RoboDK station: Dexter_ER2.rdk

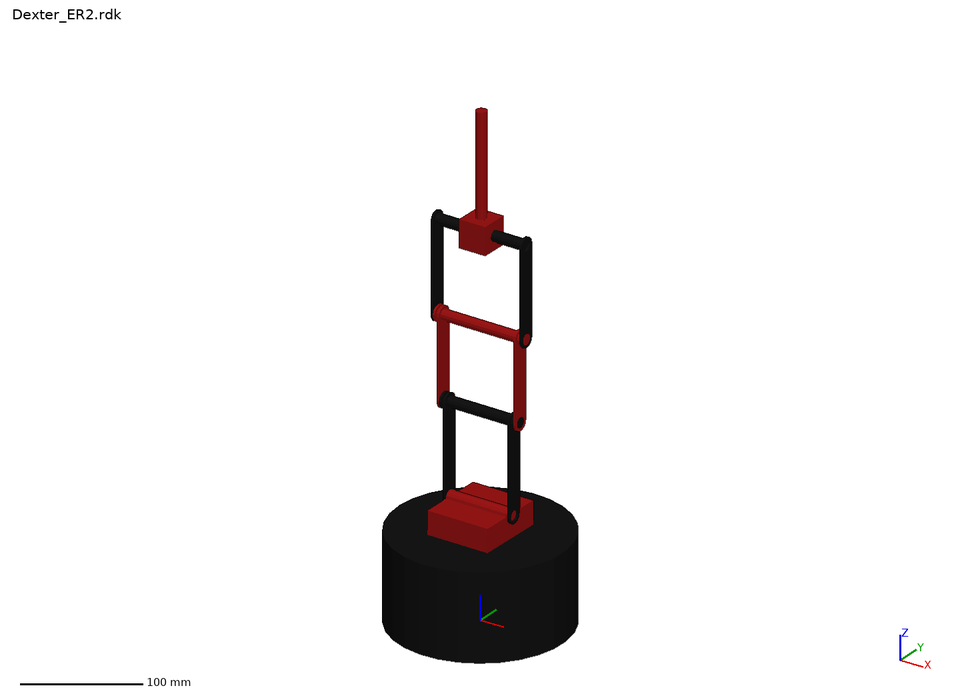
[picture v0: the station drawn from its stored meshes, robots at their saved joint values, targets as dots, program paths as lines]
Station Dexter_ER2 (saved by RoboDK 5.9.6). Poses are relative to the parent item; angles as X-Y-Z fixed-axis rotations.
  - frame Frame 1 at (0, 1000, 0) mm
    - object ER2_Fusion_baselink at (0, 0, 0) mm, size 159.5 x 159.8 x 82 mm, geometry from ER2_Fusion_baselink.step
    - object ER2_Fusion_link1 at (0, 0, 0) mm, size 64 x 65 x 37.8 mm, geometry from ER2_Fusion_link1.step
    - object ER2_Fusion_link4 at (0, 0, 0) mm, size 90 x 15 x 99.6 mm, geometry from ER2_Fusion_link4.step
    - object ER2_Fusion_ilnk5 at (0, 0, 0) mm, size 26 x 26 x 123 mm, geometry from ER2_Fusion_ilnk5.step
      - object Tool 1 at (0, 0, 430) mm
    - object ER2_Fusion_link2 at (0, 0, 0) mm, size 78 x 15 x 100.8 mm, geometry from ER2_Fusion_link2.step
    - object ER2_Fusion_link3 at (0, 0, 0) mm, size 90 x 15 x 91.8 mm, geometry from ER2_Fusion_link3.step
